FUNCTION_BLOCK FB_TCP_IP_SocketListen
VAR_INPUT
	sSrvNetId: T_AmsNetId;
	sLocalHost: T_IPv4Addr;
	nLocalPort: UDINT;
	bListen: BOOL;		//	1: Listen | 0: Stop listening, remove all existing connections
	bClose: BOOL;
	bReset: BOOL;
	TIMEOUT: TIME := T#5s;
	
END_VAR
VAR_OUTPUT
	bDone: BOOL;
	bBusy: BOOL;
	bListening: BOOL;
	hListener: Tc2_TcpIp.T_HSOCKET;
	bError: BOOL;
	nErrID: UDINT;
	sStatus: STRING(255);
	
END_VAR
VAR
	step: (eInit, eInitToListen, eListen, eWait, eClose, eClose2, eError);
	fbSocketListen: FB_SocketListen;
	fbSocketClose: FB_SocketClose;
	
	tonCaseStuck: TON;
	rtClose: R_TRIG;
	M_Close: BOOL;
	tonCloseCmdOverride: TON;
	rtReset: R_TRIG;
	M_Reset: BOOL;
	tonResetCmdOverride: TON;
	tonAutoErrorReset: TON;
	_doneSetFromCloseCase: BOOL;
	_doneSetFromListenCase: BOOL;
END_VAR

	
	rtClose(CLK:= bClose, Q=> );
	IF rtClose.Q THEN
		M_Close			:=	TRUE;
	END_IF
	tonCloseCmdOverride(IN:= M_Close, PT:= TIMEOUT + T#1S, Q=> , ET=> );
	IF tonCloseCmdOverride.Q THEN
		step		:=	eClose;
		M_Close		:=	FALSE;			
	END_IF

	rtReset(CLK:= bReset, Q=> );
	IF rtReset.Q THEN
		M_Reset			:=	TRUE;
	END_IF
	
	IF bDone AND tonResetCmdOverride.Q THEN
		step		:=	eInit;
		M_Reset		:=	FALSE;
		bDone		:=	FALSE;	
	END_IF
	tonResetCmdOverride(IN:= M_Reset, PT:= TIMEOUT + T#1S, Q=> , ET=> );
	IF tonResetCmdOverride.Q THEN
		bDone		:=	TRUE;		
	END_IF
	
	CASE step OF
	eInit:
		IF M_Close AND (NOT bReset) THEN
			step		:=	eClose;
			M_Close		:=	FALSE;
			bBusy		:=	TRUE;
			bDone		:=	FALSE;
		ELSIF bListen AND (NOT bReset) AND (NOT bClose) THEN
			step		:=	eInitToListen;		
			fbSocketListen(bExecute:= FALSE);
			fbSocketClose(bExecute:=	FALSE);
			bListening	:=	FALSE;
			bBusy		:=	TRUE;
			bDone		:=	FALSE;
		END_IF
		M_Reset			:=	FALSE;
		tonAutoErrorReset(IN:= FALSE);
		tonCaseStuck(IN:= FALSE);
		
		IF _doneSetFromCloseCase AND bDone AND NOT bClose THEN
			_doneSetFromCloseCase	:=	FALSE;
			bDone					:=	FALSE;
		END_IF
		
	eInitToListen:
		tonCaseStuck(IN:= TRUE, PT:= TIMEOUT + T#2S, Q=> , ET=> );

		fbSocketListen(
			sSrvNetId		:= sSrvNetId, 
			sLocalHost		:= sLocalHost, 
			nLocalPort		:= nLocalPort, 
			bExecute		:= TRUE, 
			tTimeout		:= TIMEOUT, 
			bBusy			=> , 
			bError			=> , 
			nErrId			=> , 
			hListener		=> hListener);		
		
		IF fbSocketListen.bError THEN
			step		:=	eError;
			nErrID		:=	fbSocketListen.nErrId;
			sStatus		:=	'FB Error: fbSocketListen | case no. eInitToListen';			
		ELSIF (fbSocketListen.bBusy) THEN
			step		:=	eListen;
			tonCaseStuck(IN:= FALSE);	
		END_IF
		
		IF tonCaseStuck.Q THEN
			IF M_Close THEN				
				step		:=	eClose;
				M_Close		:=	FALSE;
				tonCaseStuck(IN:= FALSE);
			ELSE
				step		:=	eError;
				nErrID		:=	1;
				sStatus		:=	'Custom ErrID | Case stuck: eInitToListen';
				tonCaseStuck(IN:= FALSE);	
			END_IF
		END_IF
		
	eListen:
		tonCaseStuck(IN:= TRUE, PT:= TIMEOUT + T#2S, Q=> , ET=> );

		fbSocketListen(
			sSrvNetId		:= sSrvNetId, 
			sLocalHost		:= sLocalHost, 
			nLocalPort		:= nLocalPort, 
			bExecute		:= TRUE, 
			tTimeout		:= TIMEOUT, 
			bBusy			=> , 
			bError			=> , 
			nErrId			=> , 
			hListener		=> hListener);		
		
		IF fbSocketListen.bError THEN
			step		:=	eError;
			nErrID		:=	fbSocketListen.nErrId;
			sStatus		:=	'FB Error: fbSocketListen | case no. eListen';			
		ELSIF (NOT fbSocketListen.bBusy) THEN
			fbSocketListen(bExecute:= FALSE);
			IF M_Close THEN
				step		:=	eClose;
				M_Close		:=	FALSE;
				tonCaseStuck(IN:= FALSE);
			ELSE
				step		:=	eWait;
				bListening	:=	TRUE;
				bBusy		:=	FALSE;
				bDone		:=	TRUE;
				_doneSetFromListenCase	:=	TRUE;
				tonCaseStuck(IN:= FALSE);
				bError		:=	FALSE;
				nErrID		:=	0;
				sStatus		:=	'';
			END_IF
		END_IF	

		IF tonCaseStuck.Q THEN
			IF M_Close THEN				
				step		:=	eClose;
				M_Close		:=	FALSE;
				tonCaseStuck(IN:= FALSE);
			ELSE
				step		:=	eError;
				nErrID		:=	1;
				sStatus		:=	'Custom ErrID | Case stuck: eListen';
				tonCaseStuck(IN:= FALSE);	
			END_IF				
		END_IF
		
	eWait:
		IF NOT bListen THEN
			step		:=	eClose;
			bDone		:=	FALSE;
			_doneSetFromListenCase	:=	FALSE;
		ELSIF M_Close THEN
			step		:=	eClose;	
			M_Close		:=	FALSE;
			bDone		:=	FALSE;
			_doneSetFromListenCase	:=	FALSE;
		ELSIF M_Reset THEN
			step		:=	eInit;
			bListening	:=	FALSE;
			M_Reset		:=	FALSE;
			bDone		:=	FALSE;
			_doneSetFromListenCase	:=	FALSE;	
		END_IF

		
	eClose:
		tonCaseStuck(IN:= TRUE, PT:= TIMEOUT + T#2S, Q=> , ET=> );

		bListening	:=	FALSE;
		M_Close		:=	FALSE;
		
		fbSocketClose(
			sSrvNetId		:= sSrvNetId, 
			hSocket			:= fbSocketListen.hListener, 
			bExecute		:= TRUE, 
			tTimeout		:= TIMEOUT, 
			bBusy			=> , 
			bError			=> , 
			nErrId			=> );
			
		IF fbSocketClose.bError THEN
			step		:=	eError;
			nErrID		:=	fbSocketClose.nErrId;
			sStatus		:=	'FB Error: fbSocketClose | case no. eClose';			
		ELSIF (NOT fbSocketClose.bBusy) THEN
			step		:=	eClose2;
			tonCaseStuck(IN:= FALSE);
		END_IF	
		
		IF tonCaseStuck.Q THEN
			step		:=	eError;
			nErrID		:=	1;
			sStatus		:=	'Custom ErrID | Case stuck: eClose';
			tonCaseStuck(IN:= FALSE);	
		END_IF
	
	eClose2:
		tonCaseStuck(IN:= TRUE, PT:= TIMEOUT + T#2S, Q=> , ET=> );

		fbSocketClose(
			sSrvNetId		:= sSrvNetId, 
			hSocket			:= fbSocketListen.hListener, 
			bExecute		:= TRUE, 
			tTimeout		:= TIMEOUT, 
			bBusy			=> , 
			bError			=> , 
			nErrId			=> );
			
		IF fbSocketClose.bError THEN
			step		:=	eError;
			nErrID		:=	fbSocketClose.nErrId;
			sStatus		:=	'FB Error: fbSocketClose | case no. eClose';			
		ELSIF (NOT fbSocketClose.bBusy) THEN
			fbSocketClose(bExecute:= FALSE);
			step		:=	eInit;
			bBusy		:=	FALSE;
			bDone		:=	TRUE;
			_doneSetFromCloseCase	:=	TRUE;
			tonCaseStuck(IN:= FALSE);
		END_IF	
		
		IF tonCaseStuck.Q THEN
			step		:=	eError;
			nErrID		:=	1;
			sStatus		:=	'Custom ErrID | Case stuck: eClose';
			tonCaseStuck(IN:= FALSE);	
		END_IF		
			
	eError:
		bError		:=	TRUE;
		bBusy		:=	FALSE;
		bDone		:=	FALSE;
		
		bListening	:=	FALSE;
		fbSocketListen(bExecute:= FALSE);
		fbSocketClose(bExecute:= FALSE);
		tonCaseStuck(IN:= FALSE);
		
		tonAutoErrorReset(IN:= bListen, PT:= T#5S, Q=> , ET=> );
		IF tonAutoErrorReset.Q THEN
			step	:=	eInit;
			tonAutoErrorReset(IN:= FALSE);
			
		END_IF
		
		IF M_Close THEN
			step	:=	eClose;
			M_Close	:=	FALSE;
			tonAutoErrorReset(IN:= FALSE);
			bError		:=	FALSE;
			nErrID		:=	0;
			sStatus		:=	'';
		ELSIF M_Reset THEN
			step	:=	eInit;
			M_Reset	:=	FALSE;
			tonAutoErrorReset(IN:= FALSE);
			bError		:=	FALSE;
			nErrID		:=	0;
			sStatus		:=	'';	
		END_IF
		
	END_CASE
	

	
	
	//	Calling
	fbSocketListen();
	fbSocketClose();
	tonCaseStuck();
	tonAutoErrorReset();

END_FUNCTION_BLOCK

(* stored: Version 1.1.0.1, ProductVersion 3.1.4024.13
   POU FB_TCP_IP_SocketListen: Id {0d9b34a4-f752-47ec-b73a-b47920219828}, SpecialFunc None *)
